TYPE ST_RejectReason_PK3_OUT2 :
STRUCT
	Reason	:STRING;
END_STRUCT
END_TYPE

(* stored: Version 1.1.0.1, ProductVersion 3.1.4024.13
   DUT ST_RejectReason_PK3_OUT2: Id {b0c8c034-3f69-4a22-ac68-cfdf52aeff61} *)
